PROGRAM MAIN
VAR
	nNum1 : INT ;
	nResult : INT;
	nMark : INT := 34;
	sGrade : STRING;
	
	
	
END_VAR

Act_Condition();
Act_Switch();

ACTION Act_Condition:
IF nNum1 = 1 THEN
	nResult := 1;
ELSIF nNum1 = 2 THEN
	nResult := 2;
IF nNum1 = 2 THEN
	nResult := 15;
END_IF
ELSIF nNum1 = 3 THEN
	nResult := 3;
ELSIF nNum1 = 2 THEN
	nResult := 4;
ELSE
	nResult := 10;		
END_IF
END_ACTION

ACTION Act_Switch:
CASE nMark OF
	91..100 :
	sGrade := 'A';
	81..90 :
	sGrade := 'B';
	71..80 :
	sGrade := 'C';
	61..70 :
	sGrade := 'D';
	ELSE
		sGrade := 'F';
END_CASE
END_ACTION

END_PROGRAM

(* stored: Version 1.1.0.1, ProductVersion 3.1.4024.16
   POU MAIN: Id {6d8bdcdb-1ad4-497d-822c-6d76fd70ad94}, SpecialFunc None
   Action Act_Condition: Id {d73d46f7-713d-4c96-a18d-c54b273a747b}
   Action Act_Switch: Id {f3176663-e29b-44dc-bfb1-01210f2c054f} *)
